TYPE ST_Cyl_Inputs_Outputs :
STRUCT
END_STRUCT
END_TYPE

(* stored: Version 1.1.0.1, ProductVersion 3.1.4024.6
   DUT ST_Cyl_Inputs_Outputs: Id {e0a4fe0e-a67c-0d69-05ee-371512278067} *)
